// TIA Portal V18 export
TYPE "PartCodeStruct_UDT"
// stored: IsFailsafeCompliant false
   STRUCT
      PartCode : String;   // 接收到的物料码
      PartCode_Len : Int;   // 接收到的物料码长度
      SupplierID : String[10];   // 供应商代码
      MaterialType : String[20];   // 存货编码，物料型号
      PO_ID : String[20];   // 订单编号
      BatchID : String[20];   // 批次号
      Quality : String[5];   // 数量
      Cartons : String[3];   // 箱数
      PartQuality : DInt;
   END_STRUCT;
END_TYPE
